// TIA Portal project "CONVERT_Tom_Des" (V19)

(* hardware
DEVICE "SIMATIC 1200 station_1"  S71200.Device
   slot 0: "S7-1200 rack"  Rack  V1.0
   slot 1: "PLC_1"  CPU 1214C DC/DC/DC  6ES7 214-1AG40-0XB0  V4.0
   slot 3: "AQ1 x 12 bits_1"  6ES7 232-4HA30-0XB0  V1.0
DEVICE "HMI_1"  KTP600 Basic color PN
   slot 0: "HMI"  HMI  6AV6 647-0AD11-3AX0  12.0.0.0
   slot 1: "HMI_RT_1"  KTP600 Basic color PN  6AV6 647-0AD11-3AX0  12.0.0.0
   slot 5: "IE_CP_1"  PROFINET Interface  IE_CP  V7.1.0
      slot 1: "PROFINET_Interface_1"  PROFINET Interface
         slot 1: "PORT_1"  Port  1.0.0.0
*)

// ===== PLC "PLC_1"  CPU 1214C DC/DC/DC =====

VAR_GLOBAL   // PLC tag table "Default tag table"
   "CONVERT_PB" AT %I0.0 : Bool;   // Convert Temperature N.O. Pushbutton
   "RESET_PB" AT %I0.3 : Bool;   // Data Error Reset, N.O. Pushbutton
   "ERROR_DUP_VAL" AT %Q0.0 : Bool;   // Error Indicator
   "ERROR_OVER_VAL" AT %Q0.1 : Bool;   // Data Error, Over Value
   "LL_INDC" AT %Q0.2 : Bool;   // Low Low Indicator
   "L_INDC" AT %Q0.3 : Bool;   // Low Indicator
   "M_INDC" AT %Q0.4 : Bool;   // Mid Indicator
   "H_INDC" AT %Q0.5 : Bool;   // High Indicator
   "HH_INDC" AT %Q0.6 : Bool;   // High High Indicator
END_VAR

DATA_BLOCK "Data_block_HMI"   // DB1
{ S7_Optimized_Access := 'TRUE' }
VERSION : 0.1
   VAR
      HMI_CONVERT_PB : Bool;   // HMI Convert Button
      HMI_RESET_PB : Bool;   // HMI Reset Button
      HMI_ENABLE_DISABLE : Bool;   // HMI ENABLE/DISABLE Button
   END_VAR
BEGIN
END_DATA_BLOCK

DATA_BLOCK "Data_block_Temps"   // DB2
{ S7_Optimized_Access := 'TRUE' }
VERSION : 0.1
   VAR
      C_TEMP : DInt;   // Input of Celsius Temperature
      C_TEMP_STORAGE : DInt;   // Storage of Celsius Temperature
      F_TEMP : DInt;   // Converted Fahrenheit Result
   END_VAR
BEGIN
END_DATA_BLOCK

DATA_BLOCK "Block_Convert_DB"   // DB3
{ S7_Optimized_Access := 'TRUE' }
VERSION : 0.1
// stored: InstanceOfName Block_Convert
"Block_Convert"
BEGIN
END_DATA_BLOCK

DATA_BLOCK "Block_Input_Control_DB"   // DB4
{ S7_Optimized_Access := 'TRUE' }
VERSION : 0.1
// stored: InstanceOfName Block_Input_Control
"Block_Input_Control"
BEGIN
END_DATA_BLOCK

FUNCTION_BLOCK "Block_Input_Control"   // FB1, LAD
{ S7_Optimized_Access := 'TRUE' }
VERSION : 0.1
   VAR
      ONE_SHOT_CONTROL : Bool;   // One Shot, Hardwired Panel
      HMI_ONE_SHOT_CONTROL : Bool;   // One Shot, HIM
      INTERNAL_CONVERT : Bool;   // Internal Control, Enable Convert
   END_VAR
   VAR_TEMP   // added for the SCL form of the ladder/FBD networks
      _w1 : Bool;
      _w2 : Bool;
   END_VAR
BEGIN

REGION Network 1: Internal Control, Enable Convert
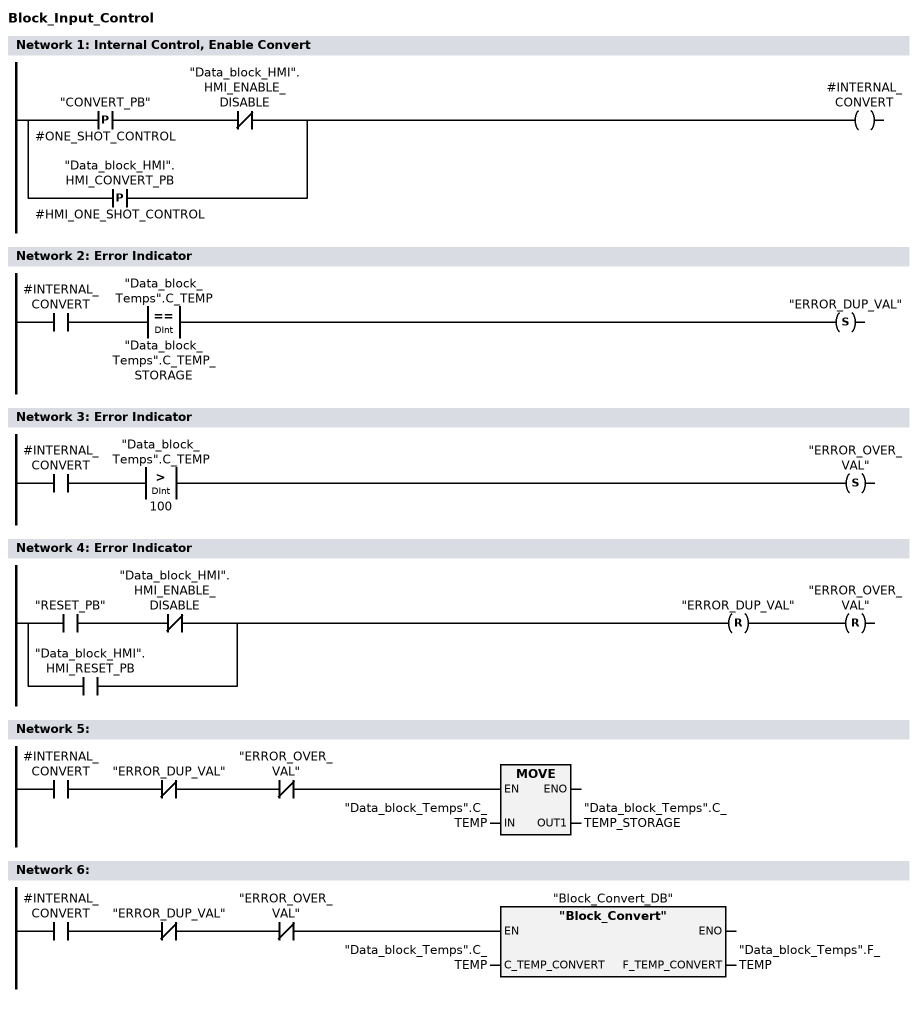
   RUNG wire#powerrail
      P_Contact(operand := "CONVERT_PB", bit := #ONE_SHOT_CONTROL)
      I_Contact( "Data_block_HMI".HMI_ENABLE_DISABLE )
      wire#w1
      Coil( #INTERNAL_CONVERT )
   END_RUNG
   RUNG wire#powerrail
      P_Contact(operand := "Data_block_HMI".HMI_CONVERT_PB, bit := #HMI_ONE_SHOT_CONTROL)
   END_RUNG wire#w1
   // the same network as SCL:
   #_w1 := "CONVERT_PB" AND NOT #ONE_SHOT_CONTROL;   // rising edge of "CONVERT_PB"
   #ONE_SHOT_CONTROL := "CONVERT_PB";
   #_w2 := "Data_block_HMI".HMI_CONVERT_PB AND NOT #HMI_ONE_SHOT_CONTROL;   // rising edge of "Data_block_HMI".HMI_CONVERT_PB
   #HMI_ONE_SHOT_CONTROL := "Data_block_HMI".HMI_CONVERT_PB;
   #INTERNAL_CONVERT := (#_w1 AND NOT "Data_block_HMI".HMI_ENABLE_DISABLE) OR #_w2;
END_REGION

REGION Network 2: Error Indicator
   RUNG wire#powerrail
      Contact( #INTERNAL_CONVERT )
      { S7_Templates := "SrcType := DInt" } EQ_Contact(in1 := "Data_block_Temps".C_TEMP, in2 := "Data_block_Temps".C_TEMP_STORAGE)
      S_Coil( "ERROR_DUP_VAL" )
   END_RUNG
   // the same network as SCL:
   IF #INTERNAL_CONVERT AND ("Data_block_Temps".C_TEMP = "Data_block_Temps".C_TEMP_STORAGE) THEN
       "ERROR_DUP_VAL" := TRUE;
   END_IF;
END_REGION

REGION Network 3: Error Indicator
   RUNG wire#powerrail
      Contact( #INTERNAL_CONVERT )
      { S7_Templates := "SrcType := DInt" } GT_Contact(in1 := "Data_block_Temps".C_TEMP, in2 := 100)
      S_Coil( "ERROR_OVER_VAL" )
   END_RUNG
   // the same network as SCL:
   IF #INTERNAL_CONVERT AND ("Data_block_Temps".C_TEMP > 100) THEN "ERROR_OVER_VAL" := TRUE; END_IF;
END_REGION

REGION Network 4: Error Indicator
   RUNG wire#powerrail
      Contact( "RESET_PB" )
      I_Contact( "Data_block_HMI".HMI_ENABLE_DISABLE )
      wire#w1
      R_Coil( "ERROR_DUP_VAL" )
      R_Coil( "ERROR_OVER_VAL" )
   END_RUNG
   RUNG wire#powerrail
      Contact( "Data_block_HMI".HMI_RESET_PB )
   END_RUNG wire#w1
   // the same network as SCL:
   IF ("RESET_PB" AND NOT "Data_block_HMI".HMI_ENABLE_DISABLE) OR "Data_block_HMI".HMI_RESET_PB THEN
       "ERROR_DUP_VAL" := FALSE;
       "ERROR_OVER_VAL" := FALSE;
   END_IF;
END_REGION

REGION Network 5
   RUNG wire#powerrail
      Contact( #INTERNAL_CONVERT )
      I_Contact( "ERROR_DUP_VAL" )
      I_Contact( "ERROR_OVER_VAL" )
      Move(in := "Data_block_Temps".C_TEMP, out1 => "Data_block_Temps".C_TEMP_STORAGE)
   END_RUNG
   // the same network as SCL:
   IF #INTERNAL_CONVERT AND NOT "ERROR_DUP_VAL" AND NOT "ERROR_OVER_VAL" THEN
       "Data_block_Temps".C_TEMP_STORAGE := "Data_block_Temps".C_TEMP;
   END_IF;
END_REGION

REGION Network 6
   RUNG wire#powerrail
      Contact( #INTERNAL_CONVERT )
      I_Contact( "ERROR_DUP_VAL" )
      I_Contact( "ERROR_OVER_VAL" )
      "Block_Convert_DB"(C_TEMP_CONVERT := "Data_block_Temps".C_TEMP, F_TEMP_CONVERT => "Data_block_Temps".F_TEMP)
   END_RUNG
   // the same network as SCL:
   IF #INTERNAL_CONVERT AND NOT "ERROR_DUP_VAL" AND NOT "ERROR_OVER_VAL" THEN
       "Block_Convert_DB"(C_TEMP_CONVERT := "Data_block_Temps".C_TEMP, F_TEMP_CONVERT => "Data_block_Temps".F_TEMP);   // "Block_Convert"
   END_IF;
END_REGION
END_FUNCTION_BLOCK

FUNCTION_BLOCK "Block_Convert"   // FB2, LAD
{ S7_Optimized_Access := 'TRUE' }
VERSION : 0.1
   VAR_INPUT
      C_TEMP_CONVERT : DInt;   // Celsius Temperature to Function Block
   END_VAR
   VAR_OUTPUT
      F_TEMP_CONVERT : DInt;   // Fahernheit Temperature From Function Block
   END_VAR
   VAR
      MUL_RESULT : DInt;   // Multipy Result
      DIV_RESULT : DInt;   // Divide Result
   END_VAR
BEGIN

REGION Network 1
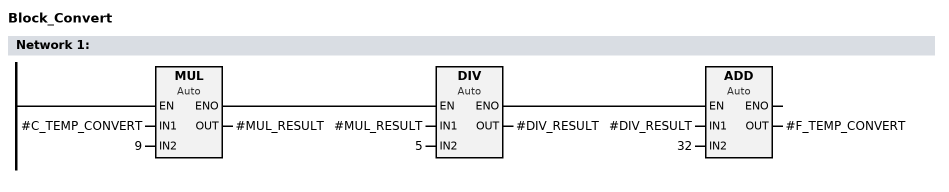
   RUNG wire#powerrail
      Mul(in1 := #C_TEMP_CONVERT, in2 := 9, out => #MUL_RESULT)
      Div(in1 := #MUL_RESULT, in2 := 5, out => #DIV_RESULT)
      Add(in1 := #DIV_RESULT, in2 := 32, out => #F_TEMP_CONVERT)
   END_RUNG
   // the same network as SCL:
   #MUL_RESULT := #C_TEMP_CONVERT * 9;
   #DIV_RESULT := #MUL_RESULT / 5;
   #F_TEMP_CONVERT := #DIV_RESULT + 32;
END_REGION
END_FUNCTION_BLOCK

FUNCTION "Block_Indicators" : Void   // FC1, LAD
{ S7_Optimized_Access := 'TRUE' }
VERSION : 0.1
BEGIN

REGION Network 1: Low Low Indicator
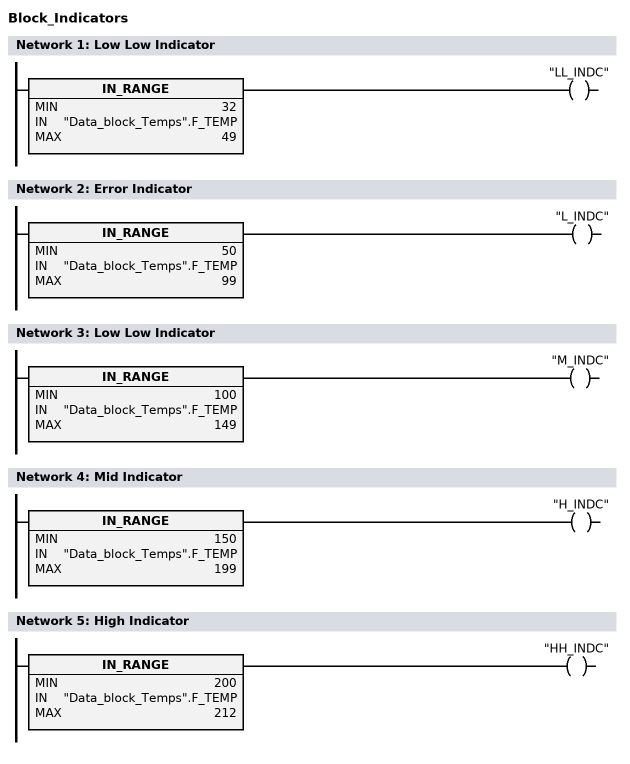
   RUNG wire#powerrail
      { S7_Templates := "SrcType := DInt" } InRange(min := 32, in := "Data_block_Temps".F_TEMP, max := 49)
      Coil( "LL_INDC" )
   END_RUNG
   // the same network as SCL:
   "LL_INDC" := (32 <= "Data_block_Temps".F_TEMP) AND ("Data_block_Temps".F_TEMP <= 49);
END_REGION

REGION Network 2: Error Indicator
   RUNG wire#powerrail
      { S7_Templates := "SrcType := DInt" } InRange(min := 50, in := "Data_block_Temps".F_TEMP, max := 99)
      Coil( "L_INDC" )
   END_RUNG
   // the same network as SCL:
   "L_INDC" := (50 <= "Data_block_Temps".F_TEMP) AND ("Data_block_Temps".F_TEMP <= 99);
END_REGION

REGION Network 3: Low Low Indicator
   RUNG wire#powerrail
      { S7_Templates := "SrcType := DInt" } InRange(min := 100, in := "Data_block_Temps".F_TEMP, max := 149)
      Coil( "M_INDC" )
   END_RUNG
   // the same network as SCL:
   "M_INDC" := (100 <= "Data_block_Temps".F_TEMP) AND ("Data_block_Temps".F_TEMP <= 149);
END_REGION

REGION Network 4: Mid Indicator
   RUNG wire#powerrail
      { S7_Templates := "SrcType := DInt" } InRange(min := 150, in := "Data_block_Temps".F_TEMP, max := 199)
      Coil( "H_INDC" )
   END_RUNG
   // the same network as SCL:
   "H_INDC" := (150 <= "Data_block_Temps".F_TEMP) AND ("Data_block_Temps".F_TEMP <= 199);
END_REGION

REGION Network 5: High Indicator
   RUNG wire#powerrail
      { S7_Templates := "SrcType := DInt" } InRange(min := 200, in := "Data_block_Temps".F_TEMP, max := 212)
      Coil( "HH_INDC" )
   END_RUNG
   // the same network as SCL:
   "HH_INDC" := (200 <= "Data_block_Temps".F_TEMP) AND ("Data_block_Temps".F_TEMP <= 212);
END_REGION
END_FUNCTION

ORGANIZATION_BLOCK "Main"   // OB1, LAD, ProgramCycle
TITLE = "Main Program Sweep (Cycle)"
{ S7_Optimized_Access := 'TRUE' }
VERSION : 0.1
BEGIN

REGION Network 1
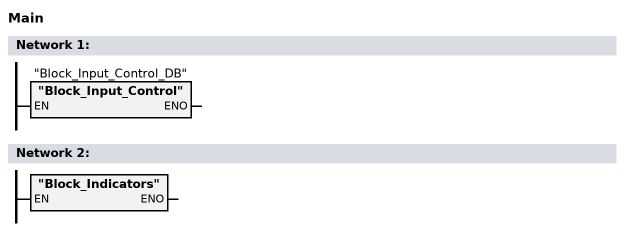
   RUNG wire#powerrail
      "Block_Input_Control_DB"()
   END_RUNG
   // the same network as SCL:
   "Block_Input_Control_DB"();   // "Block_Input_Control"
END_REGION

REGION Network 2
   RUNG wire#powerrail
      "Block_Indicators"()
   END_RUNG
   // the same network as SCL:
   "Block_Indicators"();
END_REGION
END_ORGANIZATION_BLOCK

(* ===== HMI "HMI_RT_1" =====
system functions are stored by id; their names below are inferred from use
connection "HMI_connection": ETHERNET, SMART_S7_1200_OMS

HMI tags "Default tag table"
   "HH_INDC" : Bool = PLC HH_INDC AT %Q0.6, 1 s
   "ERROR_DUP_VAL" : Bool = PLC ERROR_DUP_VAL AT %Q0.0, 1 s
   "ERROR_OVER_VAL" : Bool = PLC ERROR_OVER_VAL AT %Q0.1, 1 s
   "H_INDC" : Bool = PLC H_INDC AT %Q0.5, 1 s
   "M_INDC" : Bool = PLC M_INDC AT %Q0.4, 1 s
   "L_INDC" : Bool = PLC L_INDC AT %Q0.3, 1 s
   "LL_INDC" : Bool = PLC LL_INDC AT %Q0.2, 1 s
   "Data_block_Temps_C_TEMP" : DInt = PLC Data_block_Temps.C_TEMP, 1 s
   "Data_block_HMI_RESET_PB" : Bool = PLC Data_block_HMI.HMI_RESET_PB, 1 s
   "Data_block_HMI_CONVERT_PB" : Bool = PLC Data_block_HMI.HMI_CONVERT_PB, 1 s
   "Data_block_Temps_F_TEMP" : DInt = PLC Data_block_Temps.F_TEMP, 1 s
   "Data_block_HMI_HMI_ENABLE_DISABLE" : Bool = PLC Data_block_HMI.HMI_ENABLE_DISABLE, 1 s

Template "Template_1" 320x240
   Button "Template_" at 267,201 size 51x37; TextOff 'ExitRuntime'; PictureOff "ExitRuntime_HMI_1"; PictureOn "ExitRuntime_HMI_1"
      on Release: StopRuntime(0)

screen "Root screen" 320x240, template "Template_1"
   Softkey "Softkey_F6" at 266,202 size 53x38
      on KeyDown: StopRuntime(0)
   Button "Button_1" at 55,28 size 210x35; TextOff 'CELSIUS INPUT'
      on Release: ActivateScreen("Celsius_Input", 0)
   Button "Button_2" at 55,81 size 210x35; TextOff 'FAHRENHEIT PROCESS VALUE'
      on Release: ActivateScreen("Fahrenheit_Value", 0)
   Button "Button_3" at 55,135 size 210x35; TextOff 'MAINTENANCE'
      on Release: ActivateScreen("Maintenance", 0)

screen "Celsius_Input" 320x240, template "Template_2"
   GraphicView "Graphic view_1" at 188,7 size 120x186; Picture "Panel F Ind"
   GraphicView "Graphic view_2" at 5,7 size 183x93; Picture "Panel F Hoz"
   GraphicView "Graphic view_3" at 5,100 size 183x93; Picture "Panel F Hoz"
   GraphicView "Graphic view_4" at 199,41 size 97x37; Picture "Ind Error"
      Visibility <- "ERROR_DUP_VAL"
   GraphicView "Graphic view_5" at 199,41 size 96x36; Picture "Ind No Error"
      Visibility <- "ERROR_DUP_VAL"
   Button "Button_1" at 200,149 size 96x31; TextOff 'RESET'
      on Press: SetBit("Data_block_HMI_RESET_PB")
      on Release: ResetBit("Data_block_HMI_RESET_PB")
   GraphicView "Graphic view_6" at 199,101 size 97x37; Picture "Ind Error"
      Visibility <- "ERROR_OVER_VAL"
   GraphicView "Graphic view_7" at 199,101 size 96x36; Picture "Ind No Error"
      Visibility <- "ERROR_OVER_VAL"
   TextField "Text field_1" at 213,21 size 71x18; Text 'DUPLICATE'
   TextField "Text field_2" at 208,81 size 81x18; Text 'OVER VALUE'
   Button "Button_2" at 19,61 size 159x26; TextOff 'CONVERT'
      on Press: SetBit("Data_block_HMI_CONVERT_PB")
      on Release: ResetBit("Data_block_HMI_CONVERT_PB")
   IOField "I/O field_1" at 93,21 size 70x33; FormatPattern 999
      Visibility <- "Data_block_HMI_HMI_ENABLE_DISABLE"
      ProcessValue <- "Data_block_Temps_C_TEMP"
   TextField "Text field_3" at 26,21 size 53x34; Text 'CELSIUS INPUT'
   IOField "I/O field_2" at 63,141 size 70x33; FormatPattern 999
      ProcessValue <- "Data_block_Temps_F_TEMP"
   TextField "Text field_4" at 35,115 size 124x18; Text 'FAHRENHEIT VALUE'

screen "Fahrenheit_Value" 320x240, template "Template_3"
   TextField "Text field_2" at 126,33 size 68x16; Text 'HIGH HIGH'
   TextField "Text field_3" at 143,62 size 33x16; Text 'HIGH'
   TextField "Text field_4" at 146,94 size 27x16; Text 'MID'
   TextField "Text field_5" at 145,125 size 30x16; Text 'LOW'
   TextField "Text field_6" at 129,157 size 62x16; Text 'LOW LOW'
   GraphicView "Graphic view_3" at 205,13 size 82x181; Picture "Panel F Bar_1"
   GraphicView "Graphic view_1" at 32,13 size 82x181; Picture "Panel F Bar_1"
   Bar "Bar_1" at 37,22 size 62x164; Unit °F; MinimumValue 0; MaximumValue 220
      ProcessValue <- "Data_block_Temps_F_TEMP"
   TextField "Text field_1" at 133,0 size 55x20; Text 'RANGE'
   Rectangle "Rectangle_1" at 217,28 size 60x25
      Visibility <- "HH_INDC"
   Rectangle "Rectangle_2" at 217,59 size 60x25
      Visibility <- "H_INDC"
   Rectangle "Rectangle_3" at 217,90 size 60x25
      Visibility <- "M_INDC"
   Rectangle "Rectangle_4" at 217,121 size 60x25
      Visibility <- "L_INDC"
   Rectangle "Rectangle_5" at 217,153 size 60x25
      Visibility <- "LL_INDC"
   Group "Group" at 126,33 size 68x140

Template "Template_2" 320x240
   Button "Template_" at 267,201 size 51x37; TextOff 'ExitRuntime'; PictureOff "ExitRuntime_HMI_1"; PictureOn "ExitRuntime_HMI_1"
      on Release: StopRuntime(0)
   Button "Template_3" at 107,201 size 51x37; TextOff 'RANGE'
      on Release: ActivateScreen("Fahrenheit_Value", 0)
   Button "Template_5" at 1,201 size 51x37; TextOff 'MAIN'
      on Release: ActivateScreen("Root screen", 0)
   Button "Template_4" at 54,201 size 51x37; TextOff 'INPUT'
   Button "Template_1" at 160,201 size 51x37; TextOff 'MAINT.'
      on Release: ActivateScreen("Maintenance", 0)

Template "Template_3" 320x240
   Button "Template_" at 267,201 size 51x37; TextOff 'ExitRuntime'; PictureOff "ExitRuntime_HMI_1"; PictureOn "ExitRuntime_HMI_1"
      on Release: StopRuntime(0)
   Button "Template_4" at 54,201 size 51x37; TextOff 'INPUT'
      on Release: ActivateScreen("Celsius_Input", 0)
   Button "Template_5" at 1,201 size 51x37; TextOff 'MAIN'
      on Release: ActivateScreen("Root screen", 0)
   Button "Template_3" at 107,201 size 51x37; TextOff 'RANGE'
   Button "Template_1" at 160,201 size 51x37; TextOff 'MAINT.'
      on Release: ActivateScreen("Maintenance", 0)

screen "Maintenance" 320x240, template "Template_4"
   Switch "Switch_1" at 40,63 size 241x38; CaptionText 'Switch'; TextOff 'HARDWIRED PANEL ENABLED'; TextOn 'HARDWIRED PANEL DISABLED'
      ProcessValue <- "Data_block_HMI_HMI_ENABLE_DISABLE"

Template "Template_4" 320x240
   Button "Template_4" at 54,201 size 51x37; TextOff 'INPUT'
      on Release: ActivateScreen("Celsius_Input", 0)
   Button "Template_5" at 1,201 size 51x37; TextOff 'MAIN'
      on Release: ActivateScreen("Root screen", 0)
   Button "Template_3" at 107,201 size 51x37; TextOff 'RANGE'
      on Release: ActivateScreen("Fahrenheit_Value", 0)
   Button "Template_1" at 160,201 size 51x37; TextOff 'MAINT.'
*)